//==================================================================================================
//								RJM Maszyny sp. z o.o.
//									13.05.2022
//	Obsługa alarmów gromadzeniedanych o wystąpieniu i archiwizacja
// 	v1.0	|| TC v 3.1.4024.22		|| - pierwsza wersja
//==================================================================================================
FUNCTION_BLOCK FB_ObslugaAlarmow
VAR_INPUT
	arrTablicaZdarzen						: REFERENCE TO ;
END_VAR
VAR_OUTPUT
END_VAR
VAR
END_VAR

END_FUNCTION_BLOCK

(* stored: Version 1.1.0.1, ProductVersion 3.1.4024.11
   POU FB_ObslugaAlarmow: Id {602305fb-aa33-468a-a853-cee02f62e304}, SpecialFunc None *)
